PROGRAM main
VAR_INPUT
	X0 : bool;
END_VAR

VAR_OUTPUT
	Y0 : bool;
END_VAR

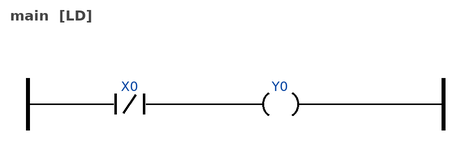
(* LD diagram, written out as Structured Text *)
Y0 := NOT X0;
END_PROGRAM
